(* PLC project BlogProject.project, CODESYS CODESYS V3.5 SP14 Patch 3 *)
(* stored: creationDateTime 2021-10-07T21:02:42.6996028, modificationDateTime 2021-10-07T20:40:20.1109198 *)

TYPE udtSystem : STRUCT
  eCurrentState : enumState;
  arTransactions : ARRAY[0..9] OF udtTransition;
END_STRUCT;
END_TYPE
